PROGRAM MAIN
VAR
		//cmt1
		btest_1:BOOL;
	btest_2: BOOL;
		
END_VAR

END_PROGRAM

(* stored: Version 1.1.0.1, ProductVersion 3.1.4024.11
   POU MAIN: Id {1f4e1dbe-6536-433b-aa85-c20dffd35be3}, SpecialFunc None *)
